TYPE "rxRecordWritePub"
TITLE = {"version":"v1.0","author":"cyanezf","family":"core/fieldbus/lldx","status":"current","deprecatedBy": null,"dependencies":[]}

//(*--
//# Documentation
//## Log
//| version | date | author | description |
//|:-------:|:----:|:------:|:------------|
//| v1.0 | 2022-10-12 | cyanezf | First version |
//
//## Description
//RX record write publisher
//--*)

   STRUCT
      providerStatus : Byte;   // Bit 0: 1=The communication with the other side of the bus has been established and the modules "RD READ PUB" and "LOCAL RD READ PUB" have been configured on the other side of the bus
   END_STRUCT;

END_TYPE

